FUNCTION_BLOCK F_INSERT (* insert IN2 into IN1 after the P-th character position *)
  (* Standard: 61131-3; Classification: standard function of character string *)
  (* Version 0.0, 2013-04-25, 4DIAC-IDE, 4DIAC-Consortium *)
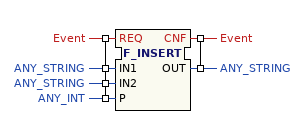
  EVENT_INPUT
    REQ WITH IN1, IN2, P; (* Service Request *)
  END_EVENT
  EVENT_OUTPUT
    CNF WITH OUT; (* Confirmation of Requested Service *)
  END_EVENT
  VAR_INPUT
    IN1 : ANY_STRING; (* input string 1 *)
    IN2 : ANY_STRING; (* input string 2 *)
    P : ANY_INT; (* insert position *)
  END_VAR
  VAR_OUTPUT
    OUT : ANY_STRING; (* string 2 inserted into string 1 at P *)
  END_VAR
END_FUNCTION_BLOCK
